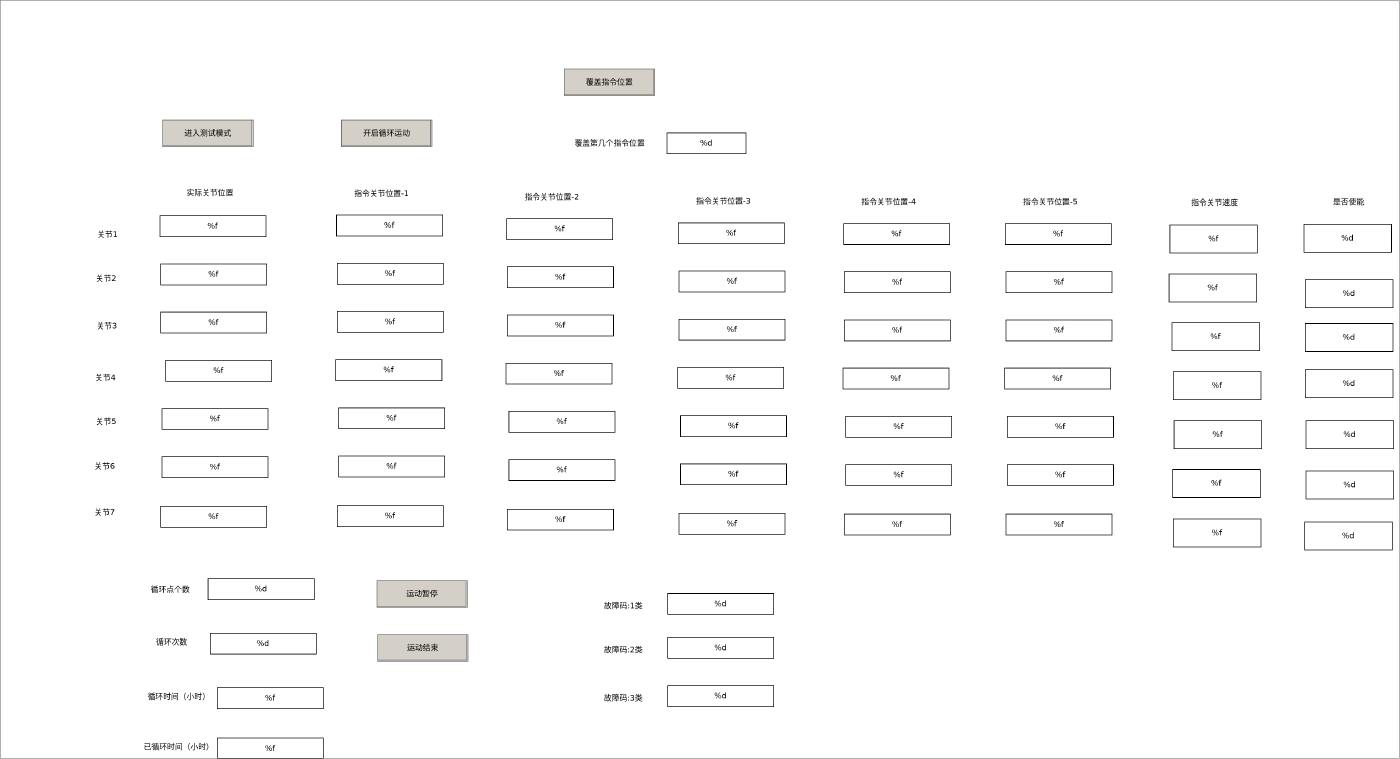
VISUALIZATION cycle_a2  // 1974x1071
    Label (221,257 150x30), "实际关节位置"
    Rectangle (225,304 150x30), "%f", text variable: g_cycleTest.m_armDHJntPos[2][1]
    Label (463,258 150x30), "指令关节位置-1"
    Button (229,169 128x38), "进入测试模式", colour toggle: g_cycleTest.m_enterCycleTestMode[2]
        toggle g_cycleTest.m_enterCycleTestMode[2]
    Button (481,169 128x38), "开启循环运动", colour toggle: g_cycleTest.m_startMotion[2]
        toggle g_cycleTest.m_startMotion[2]
    Rectangle (226,372 150x30), "%f", text variable: g_cycleTest.m_armDHJntPos[2][2]
    Rectangle (226,440 150x30), "%f", text variable: g_cycleTest.m_armDHJntPos[2][3]
    Rectangle (233,508 150x30), "%f", text variable: g_cycleTest.m_armDHJntPos[2][4]
    Rectangle (228,576 150x30), "%f", text variable: g_cycleTest.m_armDHJntPos[2][5]
    Rectangle (228,644 150x30), "%f", text variable: g_cycleTest.m_armDHJntPos[2][6]
    Rectangle (226,714 150x30), "%f", text variable: g_cycleTest.m_armDHJntPos[2][7]
    Rectangle (474,303 150x30), "%f", text variable: g_cycleTest.m_targetJntPos[2,1][1]
        OnMouseClick: write the text variable via Default
    Rectangle (475,371 150x30), "%f", text variable: g_cycleTest.m_targetJntPos[2,1][2]
        OnMouseClick: write the text variable via Default
    Rectangle (475,439 150x30), "%f", text variable: g_cycleTest.m_targetJntPos[2,1][3]
        OnMouseClick: write the text variable via Default
    Rectangle (473,507 150x30), "%f", text variable: g_cycleTest.m_targetJntPos[2,1][4]
        OnMouseClick: write the text variable via Default
    Rectangle (477,575 150x30), "%f", text variable: g_cycleTest.m_targetJntPos[2,1][5]
        OnMouseClick: write the text variable via Default
    Rectangle (477,643 150x30), "%f", text variable: g_cycleTest.m_targetJntPos[2,1][6]
        OnMouseClick: write the text variable via Default
    Rectangle (475,713 150x30), "%f", text variable: g_cycleTest.m_targetJntPos[2,1][7]
        OnMouseClick: write the text variable via Default
    Label (703,263 150x30), "指令关节位置-2"
    Rectangle (714,308 150x30), "%f", text variable: g_cycleTest.m_targetJntPos[2,2][1]
        OnMouseClick: write the text variable via Default
    Rectangle (715,376 150x30), "%f", text variable: g_cycleTest.m_targetJntPos[2,2][2]
        OnMouseClick: write the text variable via Default
    Rectangle (715,444 150x30), "%f", text variable: g_cycleTest.m_targetJntPos[2,2][3]
        OnMouseClick: write the text variable via Default
    Rectangle (713,512 150x30), "%f", text variable: g_cycleTest.m_targetJntPos[2,2][4]
        OnMouseClick: write the text variable via Default
    Rectangle (717,580 150x30), "%f", text variable: g_cycleTest.m_targetJntPos[2,2][5]
        OnMouseClick: write the text variable via Default
    Rectangle (717,648 150x30), "%f", text variable: g_cycleTest.m_targetJntPos[2,2][6]
        OnMouseClick: write the text variable via Default
    Rectangle (715,718 150x30), "%f", text variable: g_cycleTest.m_targetJntPos[2,2][7]
        OnMouseClick: write the text variable via Default
    Label (945,269 150x30), "指令关节位置-3"
    Rectangle (956,314 150x30), "%f", text variable: g_cycleTest.m_targetJntPos[2,3][1]
        OnMouseClick: write the text variable via Default
    Rectangle (957,382 150x30), "%f", text variable: g_cycleTest.m_targetJntPos[2,3][2]
        OnMouseClick: write the text variable via Default
    Rectangle (957,450 150x30), "%f", text variable: g_cycleTest.m_targetJntPos[2,3][3]
        OnMouseClick: write the text variable via Default
    Rectangle (955,518 150x30), "%f", text variable: g_cycleTest.m_targetJntPos[2,3][4]
        OnMouseClick: write the text variable via Default
    Rectangle (959,586 150x30), "%f", text variable: g_cycleTest.m_targetJntPos[2,3][5]
        OnMouseClick: write the text variable via Default
    Rectangle (959,654 150x30), "%f", text variable: g_cycleTest.m_targetJntPos[2,3][6]
        OnMouseClick: write the text variable via Default
    Rectangle (957,724 150x30), "%f", text variable: g_cycleTest.m_targetJntPos[2,3][7]
        OnMouseClick: write the text variable via Default
    Label (1178,270 150x30), "指令关节位置-4"
    Rectangle (1189,315 150x30), "%f", text variable: g_cycleTest.m_targetJntPos[2,4][1]
        OnMouseClick: write the text variable via Default
    Rectangle (1190,383 150x30), "%f", text variable: g_cycleTest.m_targetJntPos[2,4][2]
        OnMouseClick: write the text variable via Default
    Rectangle (1190,451 150x30), "%f", text variable: g_cycleTest.m_targetJntPos[2,4][3]
        OnMouseClick: write the text variable via Default
    Rectangle (1188,519 150x30), "%f", text variable: g_cycleTest.m_targetJntPos[2,4][4]
        OnMouseClick: write the text variable via Default
    Rectangle (1192,587 150x30), "%f", text variable: g_cycleTest.m_targetJntPos[2,4][5]
        OnMouseClick: write the text variable via Default
    Rectangle (1192,655 150x30), "%f", text variable: g_cycleTest.m_targetJntPos[2,4][6]
        OnMouseClick: write the text variable via Default
    Rectangle (1190,725 150x30), "%f", text variable: g_cycleTest.m_targetJntPos[2,4][7]
        OnMouseClick: write the text variable via Default
    Label (1406,270 150x30), "指令关节位置-5"
    Rectangle (1417,315 150x30), "%f", text variable: g_cycleTest.m_targetJntPos[2,5][1]
        OnMouseClick: write the text variable via Default
    Rectangle (1418,383 150x30), "%f", text variable: g_cycleTest.m_targetJntPos[2,5][2]
        OnMouseClick: write the text variable via Default
    Rectangle (1418,451 150x30), "%f", text variable: g_cycleTest.m_targetJntPos[2,5][3]
        OnMouseClick: write the text variable via Default
    Rectangle (1416,519 150x30), "%f", text variable: g_cycleTest.m_targetJntPos[2,5][4]
        OnMouseClick: write the text variable via Default
    Rectangle (1420,587 150x30), "%f", text variable: g_cycleTest.m_targetJntPos[2,5][5]
        OnMouseClick: write the text variable via Default
    Rectangle (1420,655 150x30), "%f", text variable: g_cycleTest.m_targetJntPos[2,5][6]
        OnMouseClick: write the text variable via Default
    Rectangle (1418,725 150x30), "%f", text variable: g_cycleTest.m_targetJntPos[2,5][7]
        OnMouseClick: write the text variable via Default
    Label (165,817 150x30), "循环点个数"
    Rectangle (293,816 150x30), "%d", text variable: g_cycleTest.m_pointSum[2]
        OnMouseClick: write the text variable via Default
    Rectangle (296,893 150x30), "%d", text variable: g_cycleTest.m_curCycleNum[2]
    Label (167,891 150x30), "循环次数"
    Button (531,819 128x38), "运动暂停", colour toggle: g_cycleTest.m_pause[2]
        toggle g_cycleTest.m_pause[2]
    Button (532,895 128x38), "运动结束", colour toggle: g_cycleTest.m_finish[2]
        toggle g_cycleTest.m_finish[2]
    Button (795,97 128x38), "覆盖指令位置", colour toggle: g_cycleTest.m_coverCmdPos[1]
        tap g_cycleTest.m_coverCmdPos[2]
    Rectangle (940,187 112x30), "%d", text variable: g_cycleTest.m_pntIdForCoverCmd[2]
        OnMouseClick: write the text variable via Default
    Label (787,188 145x28), "覆盖第几个指令位置"
    Label (1640,272 145x28), "指令关节速度"
    Rectangle (1649,317 124x40), "%f", text variable: g_cycleTest.m_targetJntVel[2][1]
        OnMouseClick: write the text variable via Default
    Rectangle (1648,386 124x40), "%f", text variable: g_cycleTest.m_targetJntVel[2][2]
        OnMouseClick: write the text variable via Default
    Rectangle (1652,455 124x40), "%f", text variable: g_cycleTest.m_targetJntVel[2][3]
        OnMouseClick: write the text variable via Default
    Rectangle (1654,524 124x40), "%f", text variable: g_cycleTest.m_targetJntVel[2][4]
        OnMouseClick: write the text variable via Default
    Rectangle (1655,593 124x40), "%f", text variable: g_cycleTest.m_targetJntVel[2][5]
        OnMouseClick: write the text variable via Default
    Rectangle (1653,662 124x40), "%f", text variable: g_cycleTest.m_targetJntVel[2][6]
        OnMouseClick: write the text variable via Default
    Rectangle (1654,732 124x40), "%f", text variable: g_cycleTest.m_targetJntVel[2][6]
        OnMouseClick: write the text variable via Default
    Rectangle (306,970 150x30), "%f", text variable: g_cycleTest.m_tgtCycleTime[2]
        OnMouseClick: write the text variable via Default
    Label (177,968 150x30), "循环时间（小时）"
    Rectangle (306,1041 150x30), "%f", text variable: g_cycleTest.m_curCycleTime[2]
        OnMouseClick: write the text variable via Default
    Label (177,1039 150x30), "已循环时间（小时）"
    Label (1829,271 145x28), "是否使能"
    Rectangle (1838,316 124x40), "%d", text variable: g_cycleTest.m_jntEnable[2][1]
        OnMouseClick: write the text variable via Default
    Rectangle (1840,394 124x40), "%d", text variable: g_cycleTest.m_jntEnable[2][2]
        OnMouseClick: write the text variable via Default
    Rectangle (1840,456 124x40), "%d", text variable: g_cycleTest.m_jntEnable[2][3]
        OnMouseClick: write the text variable via Default
    Rectangle (1840,521 124x40), "%d", text variable: g_cycleTest.m_jntEnable[2][4]
        OnMouseClick: write the text variable via Default
    Rectangle (1841,593 124x40), "%d", text variable: g_cycleTest.m_jntEnable[2][5]
        OnMouseClick: write the text variable via Default
    Rectangle (1841,664 124x40), "%d", text variable: g_cycleTest.m_jntEnable[2][6]
        OnMouseClick: write the text variable via Default
    Rectangle (1839,736 124x40), "%d", text variable: g_cycleTest.m_jntEnable[2][7]
        OnMouseClick: write the text variable via Default
    Label (100,313 103x36), "关节1"
    Label (98,375 103x36), "关节2"
    Label (99,442 103x36), "关节3"
    Label (97,515 103x36), "关节4"
    Label (98,577 103x36), "关节5"
    Label (96,640 103x36), "关节6"
    Label (96,705 103x36), "关节7"
    Rectangle (941,837 150x30), "%d", text variable: GVL_interactUI.g_errIdType1
        OnMouseClick: write the text variable via Default
    Label (804,840 150x30), "故障码:1类"
    Rectangle (941,899 150x30), "%d", text variable: GVL_interactUI.g_errIdType2
        OnMouseClick: write the text variable via Default
    Label (804,902 150x30), "故障码:2类"
    Rectangle (941,967 150x30), "%d", text variable: GVL_interactUI.g_errIdType3
        OnMouseClick: write the text variable via Default
    Label (804,970 150x30), "故障码:3类"
END_VISUALIZATION

(* stored: Version 1.1.0.1, ProductVersion 3.1.4024.11
   Visu cycle_a2: Id {03b103a7-77e5-4fc3-9bed-73edb8ea21ba} *)
